	16#00004441:
		F_EtherCAT_VendorIDtoString := 'Myostat Motion Control Inc.';

	16#00004567:
		F_EtherCAT_VendorIDtoString := 'Shanghai University';

	16#00004711:
		F_EtherCAT_VendorIDtoString := 'FRABA N.V.';

	16#00004957:
		F_EtherCAT_VendorIDtoString := 'INTERWORKS Co., Ltd.';

	16#00004D43:
		F_EtherCAT_VendorIDtoString := 'SKS Control OY';

	16#00005050:
		F_EtherCAT_VendorIDtoString := 'TSUZUKI DENKI CO., LTD';

	16#00005053:
		F_EtherCAT_VendorIDtoString := 'PRESTOSOLUTION Ltd.';

	16#00005257:
		F_EtherCAT_VendorIDtoString := 'Rösch & Walter Industrie-Elektronik GmbH';

	16#00005995:
		F_EtherCAT_VendorIDtoString := 'Kristl, Seibt & Co GmbH';

	16#000060C8:
		F_EtherCAT_VendorIDtoString := 'KUKA Roboter GmbH';

	(*16#000060C8: F_EtherCAT_VendorIDtoString :='KUKA Laboratories GmbH';*)
	16#00006C78:
		F_EtherCAT_VendorIDtoString := 'N.A.T. GmbH';

	16#00007595:
		F_EtherCAT_VendorIDtoString := 'LS Mecapion Co., Ltd.';

	16#00007604:
		F_EtherCAT_VendorIDtoString := 'ONTEC CO., LTD';

	16#00007715:
		F_EtherCAT_VendorIDtoString := 'Foxnum Technology Co., Ltd.';

	16#00007716:
		F_EtherCAT_VendorIDtoString := 'Kyoei Electronics Co., Ltd.';

	16#00007880:
		F_EtherCAT_VendorIDtoString := 'NISSIN SYSTEMS Co., Ltd.';

	16#00008027:
		F_EtherCAT_VendorIDtoString := 'Satyam Computer Services Limited';

	16#00008562:
		F_EtherCAT_VendorIDtoString := 'Brother Industries Ltd.';

	16#00008818:
		F_EtherCAT_VendorIDtoString := 'Shenyang Machine Tool (Group) Design Institute Co., Ltd.';

	16#000088FA:
		F_EtherCAT_VendorIDtoString := 'SIGMATEK GmbH & Co. KG';

	16#00008909:
		F_EtherCAT_VendorIDtoString := 'AIXTRON SE';

	16#00009434:
		F_EtherCAT_VendorIDtoString := 'Shenzhen Hans Motor S&T Co., Ltd.';

	16#00009555:
		F_EtherCAT_VendorIDtoString := 'Soft Servo Systems, Inc.';

	16#00009638:
		F_EtherCAT_VendorIDtoString := 'Sungrow Power Supply Co., Ltd.';

	16#00009999:
		F_EtherCAT_VendorIDtoString := 'Amoy Dynamics (Xiamen) Co., Ltd.';

	16#0000AAAA:
		F_EtherCAT_VendorIDtoString := 'HIWIN MIKROSYSTEM CORP.';

	16#0000ABBA:
		F_EtherCAT_VendorIDtoString := 'Triamec Motion AG';

	16#0000AD84:
		F_EtherCAT_VendorIDtoString := 'Topcon Precision Agriculture';

	16#0000AED0:
		F_EtherCAT_VendorIDtoString := 'ANEDO Ltd.';

	16#0000AFFE:
		F_EtherCAT_VendorIDtoString := 'VIPA Gesellschaft für Visualisierung und Prozessautomatisierung mbH';

	16#0000B0CE:
		F_EtherCAT_VendorIDtoString := 'Viveris Technologies';

	16#0000BC00:
		F_EtherCAT_VendorIDtoString := 'Brainchild Electronic Co., Ltd.';

	16#0000BEBE:
		F_EtherCAT_VendorIDtoString := 'G.D SpA';

	16#0000BEEF:
		F_EtherCAT_VendorIDtoString := 'National Radio Astronomy Observatory';

	16#0000C0DE:
		F_EtherCAT_VendorIDtoString := 'Riedl GmbH';

	16#0000CEBA:
		F_EtherCAT_VendorIDtoString := 'KEBA AG';

	16#0000DE88:
		F_EtherCAT_VendorIDtoString := 'Dalian University of Technology';

	16#0000ECA7:
		F_EtherCAT_VendorIDtoString := 'Emmission';

	16#0000EEEE:
		F_EtherCAT_VendorIDtoString := 'Willow Garage, Inc.';

	16#0000EFFE:
		F_EtherCAT_VendorIDtoString := 'Shanghai Passiontech Information Technology Co., Ltd.';

	16#0000FE09:
		F_EtherCAT_VendorIDtoString := 'Interroll Trommelmotoren GmbH';

	16#0000FEDC:
		F_EtherCAT_VendorIDtoString := 'Silica, Avnet EMG GmbH';

	16#0000FF66:
		F_EtherCAT_VendorIDtoString := 'Harbin Institute of Technology';

	16#0000FFAA:
		F_EtherCAT_VendorIDtoString := 'RB3D';

	16#0000FFFF:
		F_EtherCAT_VendorIDtoString := 'Robotiq Inc.';

	16#00010780:
		F_EtherCAT_VendorIDtoString := 'Servotecnica SpA';

	16#000144AB:
		F_EtherCAT_VendorIDtoString := 'Steinbichler Optotechnik GmbH';

	16#00051C4B:
		F_EtherCAT_VendorIDtoString := 'SICK, Inc.';

	16#000A7B00:
		F_EtherCAT_VendorIDtoString := 'Cornelius Consult';

	16#00100000:
		F_EtherCAT_VendorIDtoString := 'Shenzhen Inovance Technology Co., Ltd.';

	16#00190050:
		F_EtherCAT_VendorIDtoString := 'Kayser-Threde GmbH';

	16#00220110:
		F_EtherCAT_VendorIDtoString := 'Research and Production Plant «EKRA»';

	16#00250993:
		F_EtherCAT_VendorIDtoString := 'Manner Sensortelemetrie GmbH';

	16#00414C54:
		F_EtherCAT_VendorIDtoString := 'ALTIMA Corp.';

	16#00442656:
		F_EtherCAT_VendorIDtoString := 'D&V Electronics Ltd.';

	16#0048554B:
		F_EtherCAT_VendorIDtoString := 'Kuhnke Automation GmbH & Co. KG';

	16#00494350:
		F_EtherCAT_VendorIDtoString := 'ICP DAS Co.,Ltd.';

	16#00495254:
		F_EtherCAT_VendorIDtoString := 'IRT SA';

	16#004A4154:
		F_EtherCAT_VendorIDtoString := 'Jenaer Antriebstechnik GmbH';

	16#004d4448:
		F_EtherCAT_VendorIDtoString := 'Heidelberger Druckmaschinen AG';

	16#004D4543:
		F_EtherCAT_VendorIDtoString := 'Mecalc PTY Limited';

	16#004F524D:
		F_EtherCAT_VendorIDtoString := 'ORMEC Systems Corp.';

	16#00505349:
		F_EtherCAT_VendorIDtoString := 'Paul Scherrer Institut';

	16#00534543:
		F_EtherCAT_VendorIDtoString := 'Samsung Electronics Co. Ltd.';

	16#00577800:
		F_EtherCAT_VendorIDtoString := 'Inca Digital Printers Limited';

	16#00616978:
		F_EtherCAT_VendorIDtoString := 'aixcon PowerSystems GmbH';

	16#00706E74:
		F_EtherCAT_VendorIDtoString := 'PONUTech';

	16#00AAAAAA:
		F_EtherCAT_VendorIDtoString := 'Altera Corporation';

	(*16#00AAAAAA: F_EtherCAT_VendorIDtoString :='Altera Europe Limited';*)
	16#00ABA1EC:
		F_EtherCAT_VendorIDtoString := 'abatec group ag';

	16#00ACCE55:
		F_EtherCAT_VendorIDtoString := 'enders Ingenieure GmbH';

	16#00AE4B4B:
		F_EtherCAT_VendorIDtoString := 'KK-electronic a/s';

	16#00C0FFEE:
		F_EtherCAT_VendorIDtoString := 'Moog Animatics';

	16#00CE7C21:
		F_EtherCAT_VendorIDtoString := 'China Electronics Technology Group Corporation, No. 21 Research Institute';

	16#00DEADBF:
		F_EtherCAT_VendorIDtoString := 'Shanghai xPartner Robotics Co.,Ltd.';

	16#00E50E50:
		F_EtherCAT_VendorIDtoString := 'ESO, European Southern Observatory';

	16#00F1F1F1:
		F_EtherCAT_VendorIDtoString := 'Williams Grand Prix Engineering Limited';

	16#01000001:
		F_EtherCAT_VendorIDtoString := 'Arlington Laboratory Corporation';

	16#01000056:
		F_EtherCAT_VendorIDtoString := 'SICK AG';

	16#01000089:
		F_EtherCAT_VendorIDtoString := 'Parker Hannifin SpA - S.B.C.';

	16#010000E8:
		F_EtherCAT_VendorIDtoString := 'Balluff GmbH';

	16#01000331:
		F_EtherCAT_VendorIDtoString := 'SHANGHAI SANY SCIENCE & TECHNOLOGY CO., LTD';

	16#012EBC73:
		F_EtherCAT_VendorIDtoString := 'TIME GROUP Inc.';

	16#01ABCDEF:
		F_EtherCAT_VendorIDtoString := 'Ma.Vi. srl';

	16#02000089:
		F_EtherCAT_VendorIDtoString := 'Parker Hannifin GmbH - EME';

	16#0200008D:
		F_EtherCAT_VendorIDtoString := 'Danfoss Drives A/S';

	16#02000331:
		F_EtherCAT_VendorIDtoString := 'SHANGHAI SANY SCIENCE & TECHNOLOGY CO., LTD';

	16#03000089:
		F_EtherCAT_VendorIDtoString := 'Parker Hannifin GmbH - EME';

	16#0300008D:
		F_EtherCAT_VendorIDtoString := 'Danfoss GmbH';

	16#04000089:
		F_EtherCAT_VendorIDtoString := 'Parker Hannifin Ltd.';

	16#0505ABCD:
		F_EtherCAT_VendorIDtoString := 'A.L.L. Lasersysteme GmbH';

	16#06402200:
		F_EtherCAT_VendorIDtoString := 'L-3 Communications, Communication Systems - West';

	16#06958326:
		F_EtherCAT_VendorIDtoString := 'BNT';

	16#07770777:
		F_EtherCAT_VendorIDtoString := 'Japan Radio Co., Ltd.';

	16#0800005A:
		F_EtherCAT_VendorIDtoString := 'Schneider Electric SA';

	16#08000089:
		F_EtherCAT_VendorIDtoString := 'Parker Hannifin GmbH';

	16#09000089:
		F_EtherCAT_VendorIDtoString := 'Parker Hannifin Corporation';

	16#0A5D0000:
		F_EtherCAT_VendorIDtoString := 'Advanced Systems Development BVBA';

	16#0C044BAC:
		F_EtherCAT_VendorIDtoString := 'Compac Sorting Equipment Ltd.';

	16#0FA00000:
		F_EtherCAT_VendorIDtoString := 'FAS Technology Co., Ltd.';

	16#0FFF8888:
		F_EtherCAT_VendorIDtoString := 'GSK CNC EQUIPMENT CO., LTD.';

	16#10000000:
		F_EtherCAT_VendorIDtoString := 'SONOTRONIC Nagel GmbH';

	16#10000002:
		F_EtherCAT_VendorIDtoString := 'Beckhoff Automation GmbH';

	16#10000004:
		F_EtherCAT_VendorIDtoString := 'ED Co., Ltd';

	16#10000031:
		F_EtherCAT_VendorIDtoString := 'SHANGHAI SANY SCIENCE & TECHNOLOGY CO., LTD';

	16#10000331:
		F_EtherCAT_VendorIDtoString := 'SHANGHAI SANY SCIENCE & TECHNOLOGY CO., LTD';

	16#12345678:
		F_EtherCAT_VendorIDtoString := 'GA Drilling, Ltd.';

	16#14533417:
		F_EtherCAT_VendorIDtoString := 'Manar Sistem Ltd.';

	16#17072003:
		F_EtherCAT_VendorIDtoString := 'METTEM-Specautomatic Ltd.';

	16#19491001:
		F_EtherCAT_VendorIDtoString := 'Tsinghua University, Department of Electronic Engineering';

	16#19821130:
		F_EtherCAT_VendorIDtoString := 'Control Z Corporation';

	16#19861230:
		F_EtherCAT_VendorIDtoString := 'Shanghai Damon Logistics Technology Co.,LTD';

	16#1BA90762:
		F_EtherCAT_VendorIDtoString := 'iba AG';

	16#20041961:
		F_EtherCAT_VendorIDtoString := 'Hengstler GmbH';

	16#20422B4C:
		F_EtherCAT_VendorIDtoString := 'Lenord Bauer & Co.GmbH';

	16#20494154:
		F_EtherCAT_VendorIDtoString := 'Universität Bremen, Institut für Automatisierungstechnik (IAT)';

	16#21494256:
		F_EtherCAT_VendorIDtoString := 'IBV - Echtzeit- und Embedded GmbH & Co. KG';

	16#22222222:
		F_EtherCAT_VendorIDtoString := 'Shanghai Cohere Electronics Technology Co., Ltd.';

	16#23091861:
		F_EtherCAT_VendorIDtoString := 'Robert Bosch GmbH';

	16#26262626:
		F_EtherCAT_VendorIDtoString := 'APDISAR (Association pour la Promotion et le Développement de l’Ecole D’Ingénieurs ESISAR)';

	16#26376345:
		F_EtherCAT_VendorIDtoString := 'Convex Co., Ltd.';

	16#2E000000:
		F_EtherCAT_VendorIDtoString := 'X2E GmbH';

	16#30000331:
		F_EtherCAT_VendorIDtoString := 'SHANGHAI SANY SCIENCE & TECHNOLOGY CO., LTD';

	16#31313131:
		F_EtherCAT_VendorIDtoString := 'Sany Intelligent Control Equipment';

	16#31393633:
		F_EtherCAT_VendorIDtoString := 'Technische Universität Darmstadt, Institut für Elektromechanische Konstruktionen';

	16#314d4b54:
		F_EtherCAT_VendorIDtoString := 'MKT Systemtechnik GmbH & Co. KG';

	16#35409865:
		F_EtherCAT_VendorIDtoString := 'Korea Electronics Technology Institute';

	16#40000331:
		F_EtherCAT_VendorIDtoString := 'SHANGHAI SANY SCIENCE & TECHNOLOGY CO., LTD';

	16#40524F54:
		F_EtherCAT_VendorIDtoString := 'Red one technologies';

	16#414D4154:
		F_EtherCAT_VendorIDtoString := 'Applied Materials Inc.';

	(*16#414D4154: F_EtherCAT_VendorIDtoString :='AKT America Inc.';*)
	16#41524341:
		F_EtherCAT_VendorIDtoString := 'ARCA TECNOLOGIE srl';

	16#4156414C:
		F_EtherCAT_VendorIDtoString := 'AVAL DATA CORPORATION';

	16#42000000:
		F_EtherCAT_VendorIDtoString := 'Trust Automation Inc.';

	16#43544C42:
		F_EtherCAT_VendorIDtoString := 'Central South University of Forestry and Technology, College of Computer Science and Information Technology';

	16#44454B31:
		F_EtherCAT_VendorIDtoString := 'DEK Printing Machines Ltd.';

	16#444B465A:
		F_EtherCAT_VendorIDtoString := 'Deutsches Krebsforschungszentrum';

	16#454D5245:
		F_EtherCAT_VendorIDtoString := 'EKTECH Elektronik';

	16#46485320:
		F_EtherCAT_VendorIDtoString := 'SHF Communication Technologies AG';

	16#464D5331:
		F_EtherCAT_VendorIDtoString := 'FMS (Flexible Manufacturing System)';

	16#474F5353:
		F_EtherCAT_VendorIDtoString := 'Marcus Goßner SYSTEM SOLUTIONS';

	16#47535953:
		F_EtherCAT_VendorIDtoString := 'Grossenbacher Systeme AG';

	16#482A0000:
		F_EtherCAT_VendorIDtoString := 'Hstar Technologies Corp.';

	16#48455673:
		F_EtherCAT_VendorIDtoString := 'University of Applied Sciences Western Switzerland, Institute of Systems Engineering';

	16#4C4E5449:
		F_EtherCAT_VendorIDtoString := 'NTI AG - LinMot';

	16#4C524358:
		F_EtherCAT_VendorIDtoString := 'Lam Research Corporation';

	16#4C746C65:
		F_EtherCAT_VendorIDtoString := 'Eltromat GmbH';

	16#4D4C5431:
		F_EtherCAT_VendorIDtoString := 'MLT Micro Laser Technology GmbH';

	16#50005000:
		F_EtherCAT_VendorIDtoString := 'Technische Universität Braunschweig';

	16#50414E43:
		F_EtherCAT_VendorIDtoString := 'Power Automation GmbH';

	16#52414649:
		F_EtherCAT_VendorIDtoString := 'RAFI GmbH & Co. KG';

	16#53545A53:
		F_EtherCAT_VendorIDtoString := 'Steinbeis-Transferzentrum Systemtechnik';

	16#54455753:
		F_EtherCAT_VendorIDtoString := 'TEWS Elektronik GmbH & Co. KG';

	16#54494158:
		F_EtherCAT_VendorIDtoString := 'Timax Electronics & Machinery Ltd.';

	16#55555555:
		F_EtherCAT_VendorIDtoString := 'OLYMPUS CORPORATION';

	16#5555AAAA:
		F_EtherCAT_VendorIDtoString := 'SIASUN Robot & Automation Co., Ltd.';

	16#55AA55AA:
		F_EtherCAT_VendorIDtoString := 'Green Field Control System (I) Pvt. Ltd.';

	16#55AA55BB:
		F_EtherCAT_VendorIDtoString := 'JT3, LLC';

	16#56475454:
		F_EtherCAT_VendorIDtoString := 'Volvo Group';

	16#6167656D:
		F_EtherCAT_VendorIDtoString := 'megatec electronic GmbH';

	16#65547241:
		F_EtherCAT_VendorIDtoString := 'Arte Motion S.p.A.';

	16#66666666:
		F_EtherCAT_VendorIDtoString := 'Chinese Academy of Sciences, Institute of Optics and Electronics (IOE)';

	16#7061756C:
		F_EtherCAT_VendorIDtoString := 'PAUL Maschinenfabrik GmbH & Co.KG';

	16#77776968:
		F_EtherCAT_VendorIDtoString := 'Mesacon Messelektronik GmbH Dresden';

	16#77778888:
		F_EtherCAT_VendorIDtoString := 'Shanghai Tech Full Electric Co., Ltd.';

	16#81696189:
		F_EtherCAT_VendorIDtoString := 'Shandong University, School of Electrical Engineering';

	16#88888888:
		F_EtherCAT_VendorIDtoString := 'ScandiNova Systems AB';

	16#90646350:
		F_EtherCAT_VendorIDtoString := 'ROBOCUBETECH Co., Ltd';

	16#99998888:
		F_EtherCAT_VendorIDtoString := 'Shanghai STEP Electric Corporation';

	16#AAAA5555:
		F_EtherCAT_VendorIDtoString := 'Sunin Technology Inc.';

	16#AAAAAAAA:
		F_EtherCAT_VendorIDtoString := 'COMIZOA Co., Ltd.';

	16#AAAABBBB:
		F_EtherCAT_VendorIDtoString := 'Ruchservomotor Ltd.';

	16#AAAAFFFF:
		F_EtherCAT_VendorIDtoString := 'Dalian Jafeng Electronics Co., Ltd.';

	16#ADD1DA7A:
		F_EtherCAT_VendorIDtoString := 'ADDI-DATA GmbH';

	16#B0500001:
		F_EtherCAT_VendorIDtoString := 'Husky Injection Molding Systems Ltd.';

	16#BCDA0001:
		F_EtherCAT_VendorIDtoString := 'JINOID CO., LTD.';

	16#C0DECAFE:
		F_EtherCAT_VendorIDtoString := 'Innovasic Inc.';

	16#D4C3B2A1:
		F_EtherCAT_VendorIDtoString := 'PULOON Technology Inc.';

	16#DEADBEEF:
		F_EtherCAT_VendorIDtoString := 'Albert Handtmann Maschinenfabrik GmbH & Co. KG';

	16#DEBE50F7:
		F_EtherCAT_VendorIDtoString := 'Dewesoft d.o.o.';

ELSE
	F_EtherCAT_VendorIDtoString := 'No ID Matches.'; (*Last Update : 31/7/2013*)
END_CASE

END_FUNCTION

// Interface/I_SafetyBase
INTERFACE I_SafetyBase EXTENDS I_BaseFB

PROPERTY DependenceFB : I_BaseFB
GET
END_GET
SET
END_SET
END_PROPERTY

PROPERTY OK : BOOL
GET
END_GET
END_PROPERTY

PROPERTY SafetyReset : I_SafetyReset
SET
END_SET
END_PROPERTY

END_INTERFACE

// Interface/I_SafetyReset
INTERFACE I_SafetyReset EXTENDS I_CyclicFB

METHOD Execute
VAR_INPUT
END_VAR
END_METHOD

PROPERTY PulseDuration : TIME
SET
END_SET
END_PROPERTY

END_INTERFACE

// Interface/I_SafetySimulation
INTERFACE I_SafetySimulation EXTENDS I_SafetyBase

METHOD SimulateSafetyDiag
VAR_INPUT
	SimulationValueDiag : UINT;
END_VAR
END_METHOD

METHOD SimulateSafetyState
VAR_INPUT
	SimulationValueState : USINT;
END_VAR
END_METHOD

END_INTERFACE

// Project Information/F_GetCompany
// This function has been automatically generated from the project information.
{attribute 'signature_flag' := '1073741824'}
{attribute 'TcGenerated'}
{attribute 'no-analysis'}
FUNCTION F_GetCompany : WSTRING
VAR_INPUT
	
END_VAR

F_GetCompany := "Beckhoff Automation LLC";

END_FUNCTION

// Project Information/F_GetTitle
// This function has been automatically generated from the project information.
{attribute 'signature_flag' := '1073741824'}
{attribute 'TcGenerated'}
{attribute 'no-analysis'}
FUNCTION F_GetTitle : WSTRING
VAR_INPUT
	
END_VAR

F_GetTitle := "SPT Diagnostic";

END_FUNCTION

// Project Information/F_GetVersion
// This function has been automatically generated from the project information.
{attribute 'signature_flag' := '1073741824'}
{attribute 'TcGenerated'}
{attribute 'no-analysis'}
FUNCTION F_GetVersion : ST_LibVersion
VAR_INPUT
	
END_VAR

F_GetVersion.iMajor := 3;
F_GetVersion.iMinor := 3;
F_GetVersion.iBuild := 8;
F_GetVersion.iRevision := 0;
F_GetVersion.sVersion := '3.3.8';
F_GetVersion.nFlags := 1;

END_FUNCTION

// Safety/Safety FBs Diagnostic/Reset Functionblocks/FB_SafetyResetPulse
FUNCTION_BLOCK FB_SafetyResetPulse EXTENDS FB_CyclicFB IMPLEMENTS I_SafetyReset
VAR
	// Reset Bit to connecto to Safety
	Reset AT %Q* : BOOL;

	// Internal Variables
	TpErrorAck	: TP;
	TofErrorAck : TOF;

	// Properties
	_PulseDuration : TIME := T#100MS;
END_VAR

METHOD CyclicLogic
IF NOT _InitComplete THEN
	_InitComplete := TRUE;
	RETURN;
END_IF

// Reset Logic
TpErrorAck(PT := _PulseDuration, Q => Reset);
IF TpErrorAck.Q THEN
	TpErrorAck.IN := FALSE;
END_IF

TofErrorAck(In := TpErrorAck.Q, PT := _PulseDuration); // Block Error messages for raising and falling edge of reset signal

// Status 
_Error	 := FALSE;
_ErrorId := 0;
_Busy	 := TofErrorAck.Q;
END_METHOD

METHOD Execute
IF TpErrorAck.Q THEN
	RETURN;
END_IF

TpErrorAck.IN := TRUE;
END_METHOD

PROPERTY PulseDuration : TIME
SET
_PulseDuration := PulseDuration;
END_SET
END_PROPERTY

END_FUNCTION_BLOCK

// Safety/Safety FBs Diagnostic/FB_Component_Safety_AndOrFB
{attribute 'no_explicit_call' := 'do not call this POU directly'} 
FUNCTION_BLOCK FB_Component_Safety_AndOrFB EXTENDS FB_Component_Safety_Base

//! @summary This method serves as the entry point for all underlying FB logic
METHOD PUBLIC CyclicLogic

//! @description This method should be called cyclically by descendant function blocks by invoking <c>SUPER^.CyclicLogic()</c>.  Alternatively, the contents of this method could be reimplemented entirely in which case a call to this method would not be necessary.
IF NOT _InitComplete THEN
	_InitComplete := Initialize();
	RETURN;
END_IF

(* Main Component Signals*)
_OK		 := SUPER^.InfoData.State = E_ComponentSafetyOrAnd_State.Run;
_Busy	 := FALSE;
_ErrorId := 0;
SUPER^.CyclicLogic();
END_METHOD

//! @summary Basic component initialization logic
METHOD PROTECTED Initialize : BOOL;

//! @description This method is called by <c>CyclicLogic()</c> as required
Initialize := Super^.Initialize();
END_METHOD

END_FUNCTION_BLOCK

// Safety/Safety FBs Diagnostic/FB_Component_Safety_Base
{attribute 'no_explicit_call' := 'do not call this POU directly'}
FUNCTION_BLOCK ABSTRACT FB_Component_Safety_Base EXTENDS FB_ComponentBase IMPLEMENTS I_SafetyBase, I_SafetySimulation
VAR
	InfoData AT %I* : ST_SafetyStateDiag;

	// Reset
	ipSafetyReset : I_SafetyReset;

	// Safety Status
	ipDependenceFB : I_BaseFB; // Pointer to FB this FB is dependent on
	_OK			   : BOOL;
END_VAR

//! @summary Clears error flags and error IDs for this component
METHOD PUBLIC Reset : BOOL
_Error	 := FALSE;
_ErrorId := 0;
IF ipSafetyReset <> 0 THEN
	ipSafetyReset.Execute();
END_IF

Reset := Super^.Reset();
END_METHOD

//! @summary This method serves as the entry point for all underlying FB logic
METHOD PUBLIC CyclicLogic

//! @description This method should be called cyclically by descendant function blocks by invoking <c>SUPER^.CyclicLogic()</c>.  Alternatively, the contents of this method could be reimplemented entirely in which case a call to this method would not be necessary.
IF NOT _InitComplete THEN
	_InitComplete := Initialize();
	RETURN;
END_IF

IF ipSafetyReset <> 0 THEN
	ipSafetyReset.CyclicLogic();
END_IF

Super^.CyclicLogic();
END_METHOD

PROPERTY DependenceFB : I_BaseFB
GET
DependenceFB := ipDependenceFB;
END_GET
SET
ipDependenceFB := DependenceFB;
END_SET
END_PROPERTY

{attribute 'monitoring' := 'variable'}
PROPERTY OK : BOOL
GET
OK := _OK;
END_GET
END_PROPERTY

PROPERTY SafetyReset : I_SafetyReset
SET
ipSafetyReset := SafetyReset;
END_SET
END_PROPERTY

METHOD SimulateSafetyDiag
VAR_INPUT
	SimulationValueDiag : UINT;
END_VAR
Infodata.Diag := SimulationValueDiag;
END_METHOD

METHOD SimulateSafetyState
VAR_INPUT
	SimulationValueState : USINT;
END_VAR
Infodata.State := SimulationValueState;
END_METHOD

//! @summary Basic component initialization logic
METHOD PROTECTED Initialize : BOOL;
{analysis -22}
IF NOT _Simulate THEN
	IF NOT _Error AND (F_GetMappingStatus(ADR(InfoData), SIZEOF(InfoData)) = EplcMappingStatus.MS_Unmapped) AND NOT _Simulate THEN
		_Error := TRUE;
		TRACE('Init Failed - State not mapped to Safety!');
	END_IF

	IF _Error THEN
		RETURN;
	END_IF
END_IF

Initialize := SUPER^.Initialize();
END_METHOD

END_FUNCTION_BLOCK

// Safety/Safety FBs Diagnostic/FB_Component_Safety_ConnectionFB
{attribute 'no_explicit_call' := 'do not call this POU directly'} 
FUNCTION_BLOCK FB_Component_Safety_ConnectionFB EXTENDS FB_Component_Safety_Base
VAR
	// Alarms
	ComponentSafetyConnectionAlarms : ARRAY[1..COMPONENT_SAFETY_CONNECTION_ALARM_COUNT] OF FB_TcAlarm;
END_VAR

VAR CONSTANT
	COMPONENT_SAFETY_CONNECTION_ALARM_COUNT : UDINT := 20;
END_VAR

METHOD PROTECTED CreateEvents
VAR
END_VAR

//! @description This method is called by <c>Initialize()</c> as required
F_CreateAllEventsInClass(Alarms		:= ComponentSafetyConnectionAlarms,
						 ClassSize	:= SIZEOF(TC_EVENTS.SafetyConnection),
						 pInitEvent := ADR(TC_EVENTS.SafetyConnection.InitReferenceEvent),
						 Prefix		:= Name);

SUPER^.CreateEvents();
END_METHOD

//! Provides basic error detection and event handling for this component
METHOD PROTECTED Monitoring
VAR_INST
	DiagWord	: WORD;
	BitMaskDiag : WORD := 16#000F;
END_VAR

(*! @descriptionThis method is called cyclically by <c>CyclicLogic()</c>*)
SUPER^.Monitoring();
IF ipSafetyReset <> 0 AND_THEN ipSafetyReset.Busy THEN
	RETURN;
END_IF

BitMaskDiag := 16#000F;
DiagWord	:= TO_WORD(SUPER^.InfoData.Diag) AND BitMaskDiag;
IF (DiagWord = 1) AND NOT ComponentSafetyConnectionAlarms[E_SafetyConnection.InvalidCommand].bRaised THEN
	RaiseAlarmWithStrings(ComponentSafetyConnectionAlarms[E_SafetyConnection.InvalidCommand], '', '');
ELSIF NOT (DiagWord = 1) AND ComponentSafetyConnectionAlarms[E_SafetyConnection.InvalidCommand].bRaised THEN
	ComponentSafetyConnectionAlarms[E_SafetyConnection.InvalidCommand].Clear(0, 0);
END_IF

IF (DiagWord = 2) AND NOT ComponentSafetyConnectionAlarms[E_SafetyConnection.UnknownCommand].bRaised THEN
	RaiseAlarmWithStrings(ComponentSafetyConnectionAlarms[E_SafetyConnection.UnknownCommand], '', '');
ELSIF NOT (DiagWord = 2) AND ComponentSafetyConnectionAlarms[E_SafetyConnection.UnknownCommand].bRaised THEN
	ComponentSafetyConnectionAlarms[E_SafetyConnection.UnknownCommand].Clear(0, 0);
END_IF

IF (DiagWord = 3) AND NOT ComponentSafetyConnectionAlarms[E_SafetyConnection.InvalidConID].bRaised THEN
	RaiseAlarmWithStrings(ComponentSafetyConnectionAlarms[E_SafetyConnection.InvalidConID], '', '');
ELSIF NOT (DiagWord = 3) AND ComponentSafetyConnectionAlarms[E_SafetyConnection.InvalidConID].bRaised THEN
	ComponentSafetyConnectionAlarms[E_SafetyConnection.InvalidConID].Clear(0, 0);
END_IF

IF (DiagWord = 4) AND NOT ComponentSafetyConnectionAlarms[E_SafetyConnection.InvalidCrc].bRaised THEN
	RaiseAlarmWithStrings(ComponentSafetyConnectionAlarms[E_SafetyConnection.InvalidCrc], '', '');
ELSIF NOT (DiagWord = 4) AND ComponentSafetyConnectionAlarms[E_SafetyConnection.InvalidCrc].bRaised THEN
	ComponentSafetyConnectionAlarms[E_SafetyConnection.InvalidCrc].Clear(0, 0);
END_IF

IF (DiagWord = 5) AND NOT ComponentSafetyConnectionAlarms[E_SafetyConnection.WatchdogExpired].bRaised THEN
	RaiseAlarmWithStrings(ComponentSafetyConnectionAlarms[E_SafetyConnection.WatchdogExpired], '', '');
ELSIF NOT (DiagWord = 5) AND ComponentSafetyConnectionAlarms[E_SafetyConnection.WatchdogExpired].bRaised THEN
	ComponentSafetyConnectionAlarms[E_SafetyConnection.WatchdogExpired].Clear(0, 0);
END_IF

IF (DiagWord = 6) AND NOT ComponentSafetyConnectionAlarms[E_SafetyConnection.InvalidFSOEAddr].bRaised THEN
	RaiseAlarmWithStrings(ComponentSafetyConnectionAlarms[E_SafetyConnection.InvalidFSOEAddr], '', '');
ELSIF NOT (DiagWord = 6) AND ComponentSafetyConnectionAlarms[E_SafetyConnection.InvalidFSOEAddr].bRaised THEN
	ComponentSafetyConnectionAlarms[E_SafetyConnection.InvalidFSOEAddr].Clear(0, 0);
END_IF

IF (DiagWord = 7) AND NOT ComponentSafetyConnectionAlarms[E_SafetyConnection.InvalidData].bRaised THEN
	RaiseAlarmWithStrings(ComponentSafetyConnectionAlarms[E_SafetyConnection.InvalidData], '', '');
ELSIF NOT (DiagWord = 7) AND ComponentSafetyConnectionAlarms[E_SafetyConnection.InvalidData].bRaised THEN
	ComponentSafetyConnectionAlarms[E_SafetyConnection.InvalidData].Clear(0, 0);
END_IF

IF (DiagWord = 8) AND NOT ComponentSafetyConnectionAlarms[E_SafetyConnection.InvalidComParameterLen].bRaised THEN
	RaiseAlarmWithStrings(ComponentSafetyConnectionAlarms[E_SafetyConnection.InvalidComParameterLen], '', '');
ELSIF NOT (DiagWord = 8) AND ComponentSafetyConnectionAlarms[E_SafetyConnection.InvalidComParameterLen].bRaised THEN
	ComponentSafetyConnectionAlarms[E_SafetyConnection.InvalidComParameterLen].Clear(0, 0);
END_IF

IF (DiagWord = 9) AND NOT ComponentSafetyConnectionAlarms[E_SafetyConnection.InavlidComParameter].bRaised THEN
	RaiseAlarmWithStrings(ComponentSafetyConnectionAlarms[E_SafetyConnection.InavlidComParameter], '', '');
ELSIF NOT (DiagWord = 9) AND ComponentSafetyConnectionAlarms[E_SafetyConnection.InavlidComParameter].bRaised THEN
	ComponentSafetyConnectionAlarms[E_SafetyConnection.InavlidComParameter].Clear(0, 0);
END_IF

IF (DiagWord = 10) AND NOT ComponentSafetyConnectionAlarms[E_SafetyConnection.InvalidUserParameterLen].bRaised THEN
	RaiseAlarmWithStrings(ComponentSafetyConnectionAlarms[E_SafetyConnection.InvalidUserParameterLen], '', '');
ELSIF NOT (DiagWord = 10) AND ComponentSafetyConnectionAlarms[E_SafetyConnection.InvalidUserParameterLen].bRaised THEN
	ComponentSafetyConnectionAlarms[E_SafetyConnection.InvalidUserParameterLen].Clear(0, 0);
END_IF

IF (DiagWord = 11) AND NOT ComponentSafetyConnectionAlarms[E_SafetyConnection.InvalidUserParameter].bRaised THEN
	RaiseAlarmWithStrings(ComponentSafetyConnectionAlarms[E_SafetyConnection.InvalidUserParameter], '', '');
ELSIF NOT (DiagWord = 11) AND ComponentSafetyConnectionAlarms[E_SafetyConnection.InvalidUserParameter].bRaised THEN
	ComponentSafetyConnectionAlarms[E_SafetyConnection.InvalidUserParameter].Clear(0, 0);
END_IF

IF (DiagWord = 12) AND NOT ComponentSafetyConnectionAlarms[E_SafetyConnection.FSoEMasterReset].bRaised THEN
	RaiseAlarmWithStrings(ComponentSafetyConnectionAlarms[E_SafetyConnection.FSoEMasterReset], '', '');
ELSIF NOT (DiagWord = 12) AND ComponentSafetyConnectionAlarms[E_SafetyConnection.FSoEMasterReset].bRaised THEN
	ComponentSafetyConnectionAlarms[E_SafetyConnection.FSoEMasterReset].Clear(0, 0);
END_IF

IF (DiagWord = 13) AND NOT ComponentSafetyConnectionAlarms[E_SafetyConnection.ModuleErrorOnSlave].bRaised THEN
	RaiseAlarmWithStrings(ComponentSafetyConnectionAlarms[E_SafetyConnection.ModuleErrorOnSlave], '', '');
ELSIF NOT (DiagWord = 13) AND ComponentSafetyConnectionAlarms[E_SafetyConnection.ModuleErrorOnSlave].bRaised THEN
	ComponentSafetyConnectionAlarms[E_SafetyConnection.ModuleErrorOnSlave].Clear(0, 0);
END_IF

IF (DiagWord = 14) AND NOT ComponentSafetyConnectionAlarms[E_SafetyConnection.ModuleError].bRaised THEN
	RaiseAlarmWithStrings(ComponentSafetyConnectionAlarms[E_SafetyConnection.ModuleError], '', '');
ELSIF NOT (DiagWord = 14) AND ComponentSafetyConnectionAlarms[E_SafetyConnection.ModuleError].bRaised THEN
	ComponentSafetyConnectionAlarms[E_SafetyConnection.ModuleError].Clear(0, 0);
END_IF

IF (DiagWord = 15) AND NOT ComponentSafetyConnectionAlarms[E_SafetyConnection.SlaveNotStarted].bRaised THEN
	RaiseAlarmWithStrings(ComponentSafetyConnectionAlarms[E_SafetyConnection.SlaveNotStarted], '', '');
ELSIF NOT (DiagWord = 15) AND ComponentSafetyConnectionAlarms[E_SafetyConnection.SlaveNotStarted].bRaised THEN
	ComponentSafetyConnectionAlarms[E_SafetyConnection.SlaveNotStarted].Clear(0, 0);
END_IF

BitMaskDiag := 16#0010;
DiagWord	:= TO_WORD(SUPER^.InfoData.Diag) AND BitMaskDiag;
IF DiagWord.4 AND NOT ComponentSafetyConnectionAlarms[E_SafetyConnection.FsoESlaveError].bRaised THEN
	RaiseAlarmWithStrings(ComponentSafetyConnectionAlarms[E_SafetyConnection.FsoESlaveError], '', '');
ELSIF NOT DiagWord.4 AND ComponentSafetyConnectionAlarms[E_SafetyConnection.FsoESlaveError].bRaised THEN
	ComponentSafetyConnectionAlarms[E_SafetyConnection.FsoESlaveError].Clear(0, 0);
END_IF

BitMaskDiag := 16#0020;
DiagWord	:= TO_WORD(SUPER^.InfoData.Diag) AND BitMaskDiag;
IF DiagWord.5 AND NOT ComponentSafetyConnectionAlarms[E_SafetyConnection.FsoESlaveFailSafeValue].bRaised THEN
	RaiseAlarmWithStrings(ComponentSafetyConnectionAlarms[E_SafetyConnection.FsoESlaveFailSafeValue], '', '');
ELSIF NOT DiagWord.5 AND ComponentSafetyConnectionAlarms[E_SafetyConnection.FsoESlaveFailSafeValue].bRaised THEN
	ComponentSafetyConnectionAlarms[E_SafetyConnection.FsoESlaveFailSafeValue].Clear(0, 0);
END_IF

BitMaskDiag := 16#0040;
DiagWord	:= TO_WORD(SUPER^.InfoData.Diag) AND BitMaskDiag;
IF DiagWord.6 AND NOT ComponentSafetyConnectionAlarms[E_SafetyConnection.Startup].bRaised THEN
	RaiseAlarmWithStrings(ComponentSafetyConnectionAlarms[E_SafetyConnection.Startup], '', '');
ELSIF NOT DiagWord.6 AND ComponentSafetyConnectionAlarms[E_SafetyConnection.Startup].bRaised THEN
	ComponentSafetyConnectionAlarms[E_SafetyConnection.Startup].Clear(0, 0);
END_IF

BitMaskDiag := 16#0080;
DiagWord	:= TO_WORD(SUPER^.InfoData.Diag) AND BitMaskDiag;
IF DiagWord.7 AND NOT ComponentSafetyConnectionAlarms[E_SafetyConnection.FsoEMasterSafeValue].bRaised THEN
	RaiseAlarmWithStrings(ComponentSafetyConnectionAlarms[E_SafetyConnection.FsoEMasterSafeValue], '', '');
ELSIF NOT DiagWord.7 AND ComponentSafetyConnectionAlarms[E_SafetyConnection.FsoEMasterSafeValue].bRaised THEN
	ComponentSafetyConnectionAlarms[E_SafetyConnection.FsoEMasterSafeValue].Clear(0, 0);
END_IF

_CurrentAlarmSeverity := F_GetMaxSeverityRaised(Alarms := ComponentSafetyConnectionAlarms, CurrentSeverity := _CurrentAlarmSeverity);
END_METHOD

//! @summary Clears error flags and error IDs for this component
METHOD PUBLIC Reset : BOOL
F_ClearAllEventsInClass(ComponentSafetyConnectionAlarms);
Reset	 := SUPER^.Reset();
END_METHOD

//! @summary This method serves as the entry point for all underlying FB logic
METHOD PUBLIC CyclicLogic
//! @description This method should be called cyclically by descendant function blocks by invoking <c>SUPER^.CyclicLogic()</c>.  Alternatively, the contents of this method could be reimplemented entirely in which case a call to this method would not be necessary.
VAR
	i : UDINT;
END_VAR
IF NOT _InitComplete THEN
	_InitComplete := Initialize();
	RETURN;
END_IF

(* Main Component Signals*)
_OK		 := SUPER^.InfoData.State = E_ComponentSafetyConnection_State.Data;
_Busy	 := FALSE;
_ErrorId := SUPER^.InfoData.Diag;
SUPER^.CyclicLogic();
END_METHOD

//! @summary Basic component initialization logic
METHOD PROTECTED Initialize : BOOL;

//! @description This method is called by <c>CyclicLogic()</c> as required
Initialize := SUPER^.Initialize();
END_METHOD

END_FUNCTION_BLOCK

// Safety/Safety FBs Diagnostic/FB_Component_Safety_EdmFB
{attribute 'no_explicit_call' := 'do not call this POU directly'}
FUNCTION_BLOCK FB_Component_Safety_EdmFB EXTENDS FB_Component_Safety_Base
VAR
	// Alarms
	ComponentSafetyEDMAlarms : ARRAY[1..COMPONENT_SAFETY_EDM_ALARM_COUNT] OF FB_TcAlarm;
END_VAR

VAR CONSTANT
	COMPONENT_SAFETY_EDM_ALARM_COUNT : UDINT := 3;
END_VAR

METHOD PROTECTED CreateEvents
VAR
END_VAR

//! @description This method is called by <c>Initialize()</c> as required
F_CreateAllEventsInClass(Alarms		:= ComponentSafetyEdmAlarms,
						 ClassSize	:= SIZEOF(TC_EVENTS.SafetyEdm),
						 pInitEvent := ADR(TC_EVENTS.SafetyEdm.InitReferenceEvent),
						 Prefix		:= Name);

SUPER^.CreateEvents();
END_METHOD

//! Provides basic error detection and event handling for this component
METHOD PROTECTED Monitoring

(*! @descriptionThis method is called cyclically by <c>CyclicLogic()</c>*)
SUPER^.Monitoring();

// No error evaluation if upper Level of Safety (Group or connection) is faulted  
IF ipDependenceFB <> 0 THEN
	IF ipDependenceFB.Error THEN
		F_ClearAllEventsInClass(ComponentSafetyEdmAlarms);
		RETURN;
	END_IF
END_IF

IF ipSafetyReset <> 0 AND_THEN ipSafetyReset.Busy THEN
	RETURN;
END_IF

IF SUPER^.InfoData.Diag.0 AND NOT ComponentSafetyEdmAlarms[E_SafetyEdm.SwitchOffTime].bRaised THEN
	RaiseAlarmWithStrings(ComponentSafetyEdmAlarms[E_SafetyEdm.SwitchOffTime], '', '');
ELSIF NOT SUPER^.InfoData.Diag.0 AND ComponentSafetyEdmAlarms[E_SafetyEdm.SwitchOffTime].bRaised THEN
	ComponentSafetyEdmAlarms[E_SafetyEdm.SwitchOffTime].Clear(0, 0);
END_IF

IF SUPER^.InfoData.Diag.1 AND NOT ComponentSafetyEdmAlarms[E_SafetyEdm.SwitchOnTime].bRaised THEN
	RaiseAlarmWithStrings(ComponentSafetyEdmAlarms[E_SafetyEdm.SwitchOnTime], '', '');
ELSIF NOT SUPER^.InfoData.Diag.1 AND ComponentSafetyEdmAlarms[E_SafetyEdm.SwitchOnTime].bRaised THEN
	ComponentSafetyEdmAlarms[E_SafetyEdm.SwitchOnTime].Clear(0, 0);
END_IF

_CurrentAlarmSeverity := F_GetMaxSeverityRaised(Alarms := ComponentSafetyEdmAlarms, CurrentSeverity := _CurrentAlarmSeverity);
END_METHOD

//! @summary Clears error flags and error IDs for this component
METHOD PUBLIC Reset : BOOL
F_ClearAllEventsInClass(ComponentSafetyEDMAlarms);
Reset	 := SUPER^.Reset();
END_METHOD

//! @summary This method serves as the entry point for all underlying FB logic
METHOD PUBLIC CyclicLogic
//! @description This method should be called cyclically by descendant function blocks by invoking <c>SUPER^.CyclicLogic()</c>.  Alternatively, the contents of this method could be reimplemented entirely in which case a call to this method would not be necessary.
VAR
	i : UDINT;
END_VAR
IF NOT _InitComplete THEN
	_InitComplete := Initialize();
	RETURN;
END_IF

(* Main Component Signals*)
_OK		 := SUPER^.InfoData.State <> E_ComponentSafetyEdm_State.Error;
_Busy	 := FALSE;
_ErrorId := SUPER^.InfoData.Diag;
SUPER^.CyclicLogic();
END_METHOD

//! @summary Basic component initialization logic
METHOD PROTECTED Initialize : BOOL;

//! @description This method is called by <c>CyclicLogic()</c> as required
Initialize := Super^.Initialize();
END_METHOD

END_FUNCTION_BLOCK

// Safety/Safety FBs Diagnostic/FB_Component_Safety_EstopFB
{attribute 'no_explicit_call' := 'do not call this POU directly'}
FUNCTION_BLOCK FB_Component_Safety_EstopFB EXTENDS FB_Component_Safety_Base
VAR
	// Internal Variables
	_ActiveName : STRING := 'pressed!';

	// Alarms
	ComponentSafetyEstopAlarms : ARRAY[1..COMPONENT_SAFETY_ESTOP_ALARM_COUNT] OF FB_TcAlarm;
END_VAR

VAR CONSTANT
	COMPONENT_SAFETY_ESTOP_ALARM_COUNT : UDINT := 8;
END_VAR

METHOD PROTECTED CreateEvents
VAR
END_VAR

//! @description This method is called by <c>Initialize()</c> as required
F_CreateAllEventsInClass(Alarms		:= ComponentSafetyEstopAlarms,
						 ClassSize	:= SIZEOF(TC_EVENTS.SafetyEstop),
						 pInitEvent := ADR(TC_EVENTS.SafetyEstop.InitReferenceEvent),
						 Prefix		:= Name);

SUPER^.CreateEvents();
END_METHOD

//! Provides basic error detection and event handling for this component
METHOD PROTECTED Monitoring

(*! @descriptionThis method is called cyclically by <c>CyclicLogic()</c>*)
SUPER^.Monitoring();

// No error evaluation if upper Level of Safety (Group or connection) is faulted  
IF ipDependenceFB <> 0 THEN
	IF ipDependenceFB.Error THEN
		F_ClearAllEventsInClass(ComponentSafetyEstopAlarms);
		RETURN;
	END_IF
END_IF

IF ipSafetyReset <> 0 AND_THEN ipSafetyReset.Busy THEN
	RETURN;
END_IF

IF NOT SUPER^.OK AND NOT ComponentSafetyEstopAlarms[E_SafetyEstop.Active].bRaised THEN
	RaiseAlarmWithStrings(ComponentSafetyEstopAlarms[E_SafetyEstop.Active], _ActiveName, '');
ELSIF SUPER^.OK AND ComponentSafetyEstopAlarms[E_SafetyEstop.Active].bRaised THEN
	ComponentSafetyEstopAlarms[E_SafetyEstop.Active].Clear(0, 0);
END_IF

IF SUPER^.InfoData.Diag.0 AND NOT ComponentSafetyEstopAlarms[E_SafetyEstop.Disc1].bRaised THEN
	RaiseAlarmWithStrings(ComponentSafetyEstopAlarms[E_SafetyEstop.Disc1], '', '');
ELSIF NOT SUPER^.InfoData.Diag.0 AND ComponentSafetyEstopAlarms[E_SafetyEstop.Disc1].bRaised THEN
	ComponentSafetyEstopAlarms[E_SafetyEstop.Disc1].Clear(0, 0);
END_IF

IF SUPER^.InfoData.Diag.1 AND NOT ComponentSafetyEstopAlarms[E_SafetyEstop.Disc2].bRaised THEN
	RaiseAlarmWithStrings(ComponentSafetyEstopAlarms[E_SafetyEstop.Disc2], '', '');
ELSIF NOT SUPER^.InfoData.Diag.1 AND ComponentSafetyEstopAlarms[E_SafetyEstop.Disc2].bRaised THEN
	ComponentSafetyEstopAlarms[E_SafetyEstop.Disc2].Clear(0, 0);
END_IF

IF SUPER^.InfoData.Diag.2 AND NOT ComponentSafetyEstopAlarms[E_SafetyEstop.Disc3].bRaised THEN
	RaiseAlarmWithStrings(ComponentSafetyEstopAlarms[E_SafetyEstop.Disc3], '', '');
ELSIF NOT SUPER^.InfoData.Diag.2 AND ComponentSafetyEstopAlarms[E_SafetyEstop.Disc3].bRaised THEN
	ComponentSafetyEstopAlarms[E_SafetyEstop.Disc3].Clear(0, 0);
END_IF

IF SUPER^.InfoData.Diag.3 AND NOT ComponentSafetyEstopAlarms[E_SafetyEstop.Disc4].bRaised THEN
	RaiseAlarmWithStrings(ComponentSafetyEstopAlarms[E_SafetyEstop.Disc4], '', '');
ELSIF NOT SUPER^.InfoData.Diag.3 AND ComponentSafetyEstopAlarms[E_SafetyEstop.Disc4].bRaised THEN
	ComponentSafetyEstopAlarms[E_SafetyEstop.Disc4].Clear(0, 0);
END_IF

IF SUPER^.InfoData.Diag.4 AND NOT ComponentSafetyEstopAlarms[E_SafetyEstop.EDM1].bRaised THEN
	RaiseAlarmWithStrings(ComponentSafetyEstopAlarms[E_SafetyEstop.EDM1], '', '');
ELSIF NOT SUPER^.InfoData.Diag.4 AND ComponentSafetyEstopAlarms[E_SafetyEstop.EDM1].bRaised THEN
	ComponentSafetyEstopAlarms[E_SafetyEstop.EDM1].Clear(0, 0);
END_IF

IF SUPER^.InfoData.Diag.5 AND NOT ComponentSafetyEstopAlarms[E_SafetyEstop.EDM2].bRaised THEN
	RaiseAlarmWithStrings(ComponentSafetyEstopAlarms[E_SafetyEstop.EDM2], '', '');
ELSIF NOT SUPER^.InfoData.Diag.5 AND ComponentSafetyEstopAlarms[E_SafetyEstop.EDM2].bRaised THEN
	ComponentSafetyEstopAlarms[E_SafetyEstop.EDM2].Clear(0, 0);
END_IF

_CurrentAlarmSeverity := F_GetMaxSeverityRaised(Alarms := ComponentSafetyEstopAlarms, CurrentSeverity := _CurrentAlarmSeverity);
END_METHOD

//! @summary Clears error flags and error IDs for this component
METHOD PUBLIC Reset : BOOL
F_ClearAllEventsInClass(ComponentSafetyEstopAlarms);
Reset		  := SUPER^.Reset();
END_METHOD

//! @summary This method serves as the entry point for all underlying FB logic
METHOD PUBLIC CyclicLogic
//! @description This method should be called cyclically by descendant function blocks by invoking <c>SUPER^.CyclicLogic()</c>.  Alternatively, the contents of this method could be reimplemented entirely in which case a call to this method would not be necessary.
VAR
	i : UDINT;
END_VAR
IF NOT _InitComplete THEN
	_InitComplete := Initialize();
	RETURN;
END_IF

(* Main Component Signals*)
_OK		 := SUPER^.InfoData.State = E_ComponentSafetyEStop_State.Run;
_Busy	 := FALSE;
_ErrorId := SUPER^.InfoData.Diag;
SUPER^.CyclicLogic();
END_METHOD

PROPERTY ActiveName : String
SET
_ActiveName := ActiveName;
END_SET
END_PROPERTY

//! @summary Basic component initialization logic
METHOD PROTECTED Initialize : BOOL;

//! @description This method is called by <c>CyclicLogic()</c> as required
Initialize := SUPER^.Initialize();
END_METHOD

END_FUNCTION_BLOCK

// Safety/Safety FBs Diagnostic/FB_Component_Safety_Group
{attribute 'no_explicit_call' := 'do not call this POU directly'}
FUNCTION_BLOCK FB_Component_Safety_Group EXTENDS FB_Component_Safety_Base
VAR
	// Safety Group Connections
	Run AT %Q* : BOOL;

	// Internal Variables
	AutoFaultAck	 : TON;
	TriggerAutoReset : R_TRIG;
	ConnectionError	 : BOOL;

	// Properties
	_AutoResetConnectionFaults : BOOL;

	// Alarms
	ComponentSafetyGroupAlarms : ARRAY[1..COMPONENT_SAFETY_GROUP_ALARM_COUNT] OF FB_TcAlarm;
END_VAR

VAR CONSTANT
	COMPONENT_SAFETY_GROUP_ALARM_COUNT : UDINT := 7;
END_VAR

METHOD PROTECTED CreateEvents
VAR
END_VAR

//! @description This method is called by <c>Initialize()</c> as required
F_CreateAllEventsInClass(Alarms		:= ComponentSafetyGroupAlarms,
						 ClassSize	:= SIZEOF(TC_EVENTS.SafetyGroup),
						 pInitEvent := ADR(TC_EVENTS.SafetyGroup.InitReferenceEvent),
						 Prefix		:= Name);

SUPER^.CreateEvents();
END_METHOD

//! Provides basic error detection and event handling for this component
METHOD PROTECTED Monitoring

(*! @descriptionThis method is called cyclically by <c>CyclicLogic()</c>*)
SUPER^.Monitoring();
IF ipSafetyReset <> 0 AND_THEN ipSafetyReset.Busy THEN
	RETURN;
END_IF

IF SUPER^.InfoData.Diag = E_ComponentSafetyGroup_Diag.FbError AND NOT ComponentSafetyGroupAlarms[E_SafetyGroup.FbError].bRaised THEN
	RaiseAlarmWithStrings(ComponentSafetyGroupAlarms[E_SafetyGroup.FbError], '', '');
ELSIF SUPER^.InfoData.Diag <> E_ComponentSafetyGroup_Diag.FbError AND ComponentSafetyGroupAlarms[E_SafetyGroup.FbError].bRaised THEN
	ComponentSafetyGroupAlarms[E_SafetyGroup.FbError].Clear(0, 0);
END_IF

IF SUPER^.InfoData.Diag = E_ComponentSafetyGroup_Diag.ComError AND NOT ComponentSafetyGroupAlarms[E_SafetyGroup.ComError].bRaised THEN
	RaiseAlarmWithStrings(ComponentSafetyGroupAlarms[E_SafetyGroup.ComError], '', '');
ELSIF SUPER^.InfoData.Diag <> E_ComponentSafetyGroup_Diag.ComError AND ComponentSafetyGroupAlarms[E_SafetyGroup.ComError].bRaised THEN
	ComponentSafetyGroupAlarms[E_SafetyGroup.ComError].Clear(0, 0);
END_IF

IF SUPER^.InfoData.Diag = E_ComponentSafetyGroup_Diag.ModuleError AND NOT ComponentSafetyGroupAlarms[E_SafetyGroup.ModuleError].bRaised THEN
	RaiseAlarmWithStrings(ComponentSafetyGroupAlarms[E_SafetyGroup.ModuleError], '', '');
ELSIF SUPER^.InfoData.Diag <> E_ComponentSafetyGroup_Diag.ModuleError AND ComponentSafetyGroupAlarms[E_SafetyGroup.ModuleError].bRaised THEN
	ComponentSafetyGroupAlarms[E_SafetyGroup.ModuleError].Clear(0, 0);
END_IF

IF SUPER^.InfoData.Diag = E_ComponentSafetyGroup_Diag.CmpError AND NOT ComponentSafetyGroupAlarms[E_SafetyGroup.CmpError].bRaised THEN
	RaiseAlarmWithStrings(ComponentSafetyGroupAlarms[E_SafetyGroup.CmpError], '', '');
ELSIF SUPER^.InfoData.Diag <> E_ComponentSafetyGroup_Diag.CmpError AND ComponentSafetyGroupAlarms[E_SafetyGroup.CmpError].bRaised THEN
	ComponentSafetyGroupAlarms[E_SafetyGroup.CmpError].Clear(0, 0);
END_IF

IF SUPER^.InfoData.Diag = E_ComponentSafetyGroup_Diag.DeactiveError AND NOT ComponentSafetyGroupAlarms[E_SafetyGroup.DeactiveError].bRaised THEN
	RaiseAlarmWithStrings(ComponentSafetyGroupAlarms[E_SafetyGroup.DeactiveError], '', '');
ELSIF SUPER^.InfoData.Diag <> E_ComponentSafetyGroup_Diag.DeactiveError AND ComponentSafetyGroupAlarms[E_SafetyGroup.DeactiveError].bRaised THEN
	ComponentSafetyGroupAlarms[E_SafetyGroup.DeactiveError].Clear(0, 0);
END_IF

IF SUPER^.InfoData.Diag = E_ComponentSafetyGroup_Diag.RestartError AND NOT ComponentSafetyGroupAlarms[E_SafetyGroup.RestartError].bRaised THEN
	RaiseAlarmWithStrings(ComponentSafetyGroupAlarms[E_SafetyGroup.RestartError], '', '');
ELSIF SUPER^.InfoData.Diag <> E_ComponentSafetyGroup_Diag.RestartError AND ComponentSafetyGroupAlarms[E_SafetyGroup.RestartError].bRaised THEN
	ComponentSafetyGroupAlarms[E_SafetyGroup.RestartError].Clear(0, 0);
END_IF

_CurrentAlarmSeverity := F_GetMaxSeverityRaised(Alarms := ComponentSafetyGroupAlarms, CurrentSeverity := _CurrentAlarmSeverity);
END_METHOD

//! @summary Clears error flags and error IDs for this component
METHOD PUBLIC Reset : BOOL
F_ClearAllEventsInClass(ComponentSafetyGroupAlarms);
Reset		  := SUPER^.Reset();
END_METHOD

//! @summary This method serves as the entry point for all underlying FB logic
METHOD PUBLIC CyclicLogic
//! @description This method should be called cyclically by descendant function blocks by invoking <c>SUPER^.CyclicLogic()</c>.  Alternatively, the contents of this method could be reimplemented entirely in which case a call to this method would not be necessary.
VAR
	i : UDINT;
END_VAR
IF NOT _InitComplete THEN
	_InitComplete := Initialize();
	RETURN;
END_IF

(*Control Group Group*)
Run				:= TRUE;
ConnectionError := SUPER^.InfoData.Diag <> 0;
IF ipSafetyReset <> 0 then
	AutoFaultAck(IN := (_AutoResetConnectionFaults AND ConnectionError) AND NOT ipSafetyReset.Busy, PT := T#250MS);
	TriggerAutoReset(CLK := AutoFaultAck.Q);
	IF TriggerAutoReset.Q then
		ipSafetyReset.Execute();
	END_IF
END_IF

(* Main Component Signals*)
_OK		 := SUPER^.InfoData.State = E_ComponentSafetyGroup_State.Run;
_Busy	 := FALSE;
_ErrorId := SUPER^.InfoData.Diag;
SUPER^.CyclicLogic();
END_METHOD

PROPERTY AutoResetConnectionFaults : BOOL
GET
AutoResetConnectionFaults := _AutoResetConnectionFaults;
END_GET
SET
_AutoResetConnectionFaults := AutoResetConnectionFaults;
END_SET
END_PROPERTY

//! @summary Basic component initialization logic
METHOD PROTECTED Initialize : BOOL;

//! @description This method is called by <c>CyclicLogic()</c> as required
{analysis -22}
IF NOT _Simulate THEN
	IF NOT _Error AND (F_GetMappingStatus(ADR(Run), SIZEOF(Run)) = EplcMappingStatus.MS_Unmapped) THEN
		_Error := TRUE;
		Trace('Init Failed - Group Run not mapped to Safety!');
	END_IF

	IF NOT _Error AND ipSafetyReset = 0 THEN
		_Error := TRUE;
		Trace('Init Failed - Group requires Safety Reset FB Instance!');
	END_IF
END_IF

IF _Error THEN
	RETURN;
END_IF

Initialize := SUPER^.Initialize();
END_METHOD

END_FUNCTION_BLOCK

// Safety/Safety FBs Diagnostic/FB_Component_Safety_MonFB
{attribute 'no_explicit_call' := 'do not call this POU directly'}
FUNCTION_BLOCK FB_Component_Safety_MonFB EXTENDS FB_Component_Safety_Base
VAR
	// Alarm at Safe State
	_ActiveAlarm : BOOL	  := TRUE;
	_ActiveName	 : STRING := 'pressed!';

	// Alarms
	ComponentSafetyMonAlarms : ARRAY[1..COMPONENT_SAFETY_MON_ALARM_COUNT] OF FB_TcAlarm;
END_VAR

VAR CONSTANT
	COMPONENT_SAFETY_MON_ALARM_COUNT : UDINT := 10;
END_VAR

METHOD PROTECTED CreateEvents
VAR
END_VAR

//! @description This method is called by <c>Initialize()</c> as required
F_CreateAllEventsInClass(Alarms		:= ComponentSafetyMonAlarms,
						 ClassSize	:= SIZEOF(TC_EVENTS.SafetyMon),
						 pInitEvent := ADR(TC_EVENTS.SafetyMon.InitReferenceEvent),
						 Prefix		:= Name);

SUPER^.CreateEvents();
END_METHOD

//! Provides basic error detection and event handling for this component
METHOD PROTECTED Monitoring

(*! @descriptionThis method is called cyclically by <c>CyclicLogic()</c>*)
SUPER^.Monitoring();

// No error evaluation if upper Level of Safety (Group or connection) is faulted  
IF ipDependenceFB <> 0 THEN
	IF ipDependenceFB.Error THEN
		F_ClearAllEventsInClass(ComponentSafetyMonAlarms);
		RETURN;
	END_IF
END_IF

IF ipSafetyReset <> 0 AND_THEN ipSafetyReset.Busy THEN
	RETURN;
END_IF

IF NOT SUPER^.OK AND _ActiveAlarm AND NOT ComponentSafetyMonAlarms[E_SafetyMon.Active].bRaised THEN
	RaiseAlarmWithStrings(ComponentSafetyMonAlarms[E_SafetyMon.Active], _ActiveName, '');
ELSIF SUPER^.OK AND ComponentSafetyMonAlarms[E_SafetyMon.Active].bRaised THEN
	ComponentSafetyMonAlarms[E_SafetyMon.Active].Clear(0, 0);
END_IF

IF SUPER^.InfoData.Diag.0 AND NOT ComponentSafetyMonAlarms[E_SafetyMon.Disc1].bRaised THEN
	RaiseAlarmWithStrings(ComponentSafetyMonAlarms[E_SafetyMon.Disc1], '', '');
ELSIF NOT SUPER^.InfoData.Diag.0 AND ComponentSafetyMonAlarms[E_SafetyMon.Disc1].bRaised THEN
	ComponentSafetyMonAlarms[E_SafetyMon.Disc1].Clear(0, 0);
END_IF

IF SUPER^.InfoData.Diag.1 AND NOT ComponentSafetyMonAlarms[E_SafetyMon.Disc2].bRaised THEN
	RaiseAlarmWithStrings(ComponentSafetyMonAlarms[E_SafetyMon.Disc2], '', '');
ELSIF NOT SUPER^.InfoData.Diag.1 AND ComponentSafetyMonAlarms[E_SafetyMon.Disc2].bRaised THEN
	ComponentSafetyMonAlarms[E_SafetyMon.Disc2].Clear(0, 0);
END_IF

IF SUPER^.InfoData.Diag.3 AND NOT ComponentSafetyMonAlarms[E_SafetyMon.DiscInput].bRaised THEN
	RaiseAlarmWithStrings(ComponentSafetyMonAlarms[E_SafetyMon.DiscInput], '', '');
ELSIF NOT SUPER^.InfoData.Diag.3 AND ComponentSafetyMonAlarms[E_SafetyMon.DiscInput].bRaised THEN
	ComponentSafetyMonAlarms[E_SafetyMon.DiscInput].Clear(0, 0);
END_IF

IF SUPER^.InfoData.Diag.4 AND NOT ComponentSafetyMonAlarms[E_SafetyMon.Edm1].bRaised THEN
	RaiseAlarmWithStrings(ComponentSafetyMonAlarms[E_SafetyMon.Edm1], '', '');
ELSIF NOT SUPER^.InfoData.Diag.4 AND ComponentSafetyMonAlarms[E_SafetyMon.Edm1].bRaised THEN
	ComponentSafetyMonAlarms[E_SafetyMon.Edm1].Clear(0, 0);
END_IF

IF SUPER^.InfoData.Diag.5 AND NOT ComponentSafetyMonAlarms[E_SafetyMon.Edm2].bRaised THEN
	RaiseAlarmWithStrings(ComponentSafetyMonAlarms[E_SafetyMon.Edm2], '', '');
ELSIF NOT SUPER^.InfoData.Diag.5 AND ComponentSafetyMonAlarms[E_SafetyMon.Edm2].bRaised THEN
	ComponentSafetyMonAlarms[E_SafetyMon.Edm2].Clear(0, 0);
END_IF

IF SUPER^.InfoData.Diag.8 AND NOT ComponentSafetyMonAlarms[E_SafetyMon.Disc1Safe].bRaised THEN
	RaiseAlarmWithStrings(ComponentSafetyMonAlarms[E_SafetyMon.Disc1Safe], '', '');
ELSIF NOT SUPER^.InfoData.Diag.8 AND ComponentSafetyMonAlarms[E_SafetyMon.Disc1Safe].bRaised THEN
	ComponentSafetyMonAlarms[E_SafetyMon.Disc1Safe].Clear(0, 0);
END_IF

IF SUPER^.InfoData.Diag.9 AND NOT ComponentSafetyMonAlarms[E_SafetyMon.Disc2Safe].bRaised THEN
	RaiseAlarmWithStrings(ComponentSafetyMonAlarms[E_SafetyMon.Disc2Safe], '', '');
ELSIF NOT SUPER^.InfoData.Diag.9 AND ComponentSafetyMonAlarms[E_SafetyMon.Disc2Safe].bRaised THEN
	ComponentSafetyMonAlarms[E_SafetyMon.Disc2Safe].Clear(0, 0);
END_IF

IF SUPER^.InfoData.Diag.10 AND NOT ComponentSafetyMonAlarms[E_SafetyMon.DiscInputSafe].bRaised THEN
	RaiseAlarmWithStrings(ComponentSafetyMonAlarms[E_SafetyMon.DiscInputSafe], '', '');
ELSIF NOT SUPER^.InfoData.Diag.10 AND ComponentSafetyMonAlarms[E_SafetyMon.DiscInputSafe].bRaised THEN
	ComponentSafetyMonAlarms[E_SafetyMon.DiscInputSafe].Clear(0, 0);
END_IF

_CurrentAlarmSeverity := F_GetMaxSeverityRaised(Alarms := ComponentSafetyMonAlarms, CurrentSeverity := _CurrentAlarmSeverity);
END_METHOD

//! @summary Clears error flags and error IDs for this component
METHOD PUBLIC Reset : BOOL
F_ClearAllEventsInClass(ComponentSafetyMonAlarms);
Reset	 := SUPER^.Reset();
END_METHOD

//! @summary This method serves as the entry point for all underlying FB logic
METHOD PUBLIC CyclicLogic
//! @description This method should be called cyclically by descendant function blocks by invoking <c>SUPER^.CyclicLogic()</c>.  Alternatively, the contents of this method could be reimplemented entirely in which case a call to this method would not be necessary.
VAR
	i : UDINT;
END_VAR
IF NOT _InitComplete THEN
	_InitComplete := Initialize();
	RETURN;
END_IF

(* Main Component Signals*)
_OK		 := SUPER^.InfoData.State = E_ComponentSafetyMon_State.Run;
_Busy	 := FALSE;
_ErrorId := SUPER^.InfoData.Diag;
SUPER^.CyclicLogic();
END_METHOD

PROPERTY PUBLIC ActiveAlarm : BOOL
SET
_ActiveAlarm := ActiveAlarm;
END_SET
END_PROPERTY

PROPERTY ActiveName : String
SET
_ActiveName := ActiveName;
END_SET
END_PROPERTY

END_FUNCTION_BLOCK
